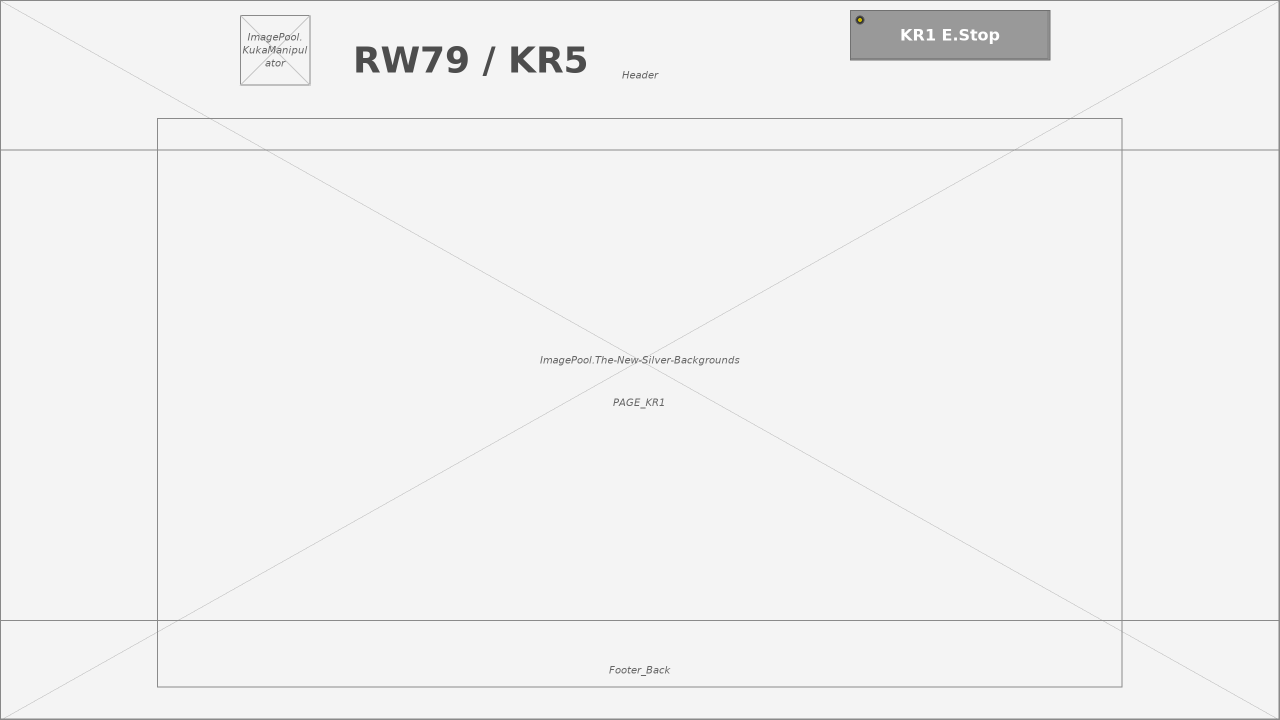
VISUALIZATION PAGE_KR1_Tab  // 1280x720
    Image (0,0 1280x720), image: ImagePool.The-New-Silver-Backgrounds
    Frame (0,620 1280x100)
        shows Footer_Back()
    Frame (0,0 1280x150)
        shows Header()
    Label (350,40 300x40), "RW79 / KR5"
    Group (850,10 200x50)
        Button (0,0 200x50), "KR1 E.Stop"
            toggle KR1.KR1_Estop
        Lamp1 (5,5 10x10), variable: KR1.KR1_Estop, style: Lamp-Lamp1-Yellow
    Image (240,15 70x70), image: ImagePool.KukaManipulator
    TabControl (157,118 965x569)
        shows PAGE_KR1()
        shows PAGE_KR1_Tab_1_100()
        shows PAGE_KR1_Tab_1_200()
        [0]: TabTitle=Main
        [1]: TabTitle=1-100
        [2]: TabTitle=100-200
END_VISUALIZATION

(* stored: Version 1.1.0.1, ProductVersion 3.1.4024.12
   Visu PAGE_KR1_Tab: Id {ca5687a6-0a32-43d4-b8c0-7e10f27352c2} *)
